// TwinCAT 3 PLC project Math
// Title: Math
// Company: TomasRompotl
// ProjectVersion: 0.0.1
// ProgramVersion: 3.1.4024.0
// project tree:
//   Point/ Point3D.TcDUT (not stored), Point2D.TcDUT (not stored)
//   Range/ IsInRangeInclusive.TcPOU, IsInRangeInclusive2D.TcPOU (not stored), IsInRangeInclusive3D.TcPOU, Range2D.TcDUT (not stored), Range3D.TcDUT (not stored), Range.TcDUT
//   Version/ Global_Version.TcGVL
// real-time tasks:
//   TASK BindingTestTask: cycle T#1ms, priority 20, ADS port 350
//   TASK PlcTask: cycle T#1ms, priority 21, ADS port 351
//   TASK PlcTask1: cycle T#1ms, priority 22, ADS port 352
//   TASK PlcTask2: cycle T#1ms, priority 23, ADS port 353
//   TASK MathTestTask: cycle T#1ms, priority 24, ADS port 354
//   TASK TimesTestsTask: cycle T#1ms, priority 25, ADS port 355

// ---- Range/Range.TcDUT
TYPE Range :
STRUCT
	Bottom : LREAL;
	Top : LREAL;
END_STRUCT
END_TYPE

// ---- Version/Global_Version.TcGVL
{attribute 'TcGenerated'}
{attribute 'no-analysis'}
{attribute 'linkalways'}
// This function has been automatically generated from the project information.
VAR_GLOBAL CONSTANT
	{attribute 'const_non_replaced'}
	stLibVersion_Math : ST_LibVersion := (iMajor := 0, iMinor := 0, iBuild := 1, iRevision := 0, nFlags := 0, sVersion := '0.0.1');
END_VAR

// ---- Range/IsInRangeInclusive.TcPOU
FUNCTION IsInRangeInclusive : BOOL
VAR_INPUT
	value : LREAL;
	range : Range;
END_VAR

IsInRangeInclusive := range.Bottom <= value AND value <= range.Top;

END_FUNCTION

// ---- Range/IsInRangeInclusive3D.TcPOU
FUNCTION IsInRangeInclusive3D : BOOL
VAR_INPUT
	point : Point3D;
	range : Range3D;
END_VAR

IsInRangeInclusive3D := 
	IsInRangeInclusive(point.X, range.X)
	AND IsInRangeInclusive(point.Y, range.Y)
	AND IsInRangeInclusive(point.Z, range.Z)
	;

END_FUNCTION
